ABB RobotStudio station: HCV_1.rsstn

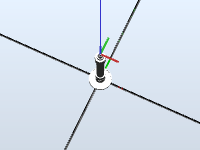
Station HCV (saved by RobotStudio 6.5.7558.2005)
Layout (positions relative to the parent item):
  - HCV [mechanism] at (0, 0, 0) mm
      TCP HCVTCP at (0, 191.01, 0) mm, rotated rx -90 ry 0 rz 0 deg
      links: HERRAMIENTA
